PROGRAM PRG_SL2L0_POWER
VAR
	fbMotion1: FB_SimMotor;
	fbMotion2: FB_SimMotor;
	fbMotion3: FB_SimMotor;
	fbMotion4: FB_SimMotor;
END_VAR

// Placeholder, standard simulated motion for all axes
fbMotion1(stMotionStage := Main.M45);
fbMotion2(stMotionStage := Main.M46);
fbMotion3(stMotionStage := Main.M47);
fbMotion4(stMotionStage := Main.M48);

END_PROGRAM

(* stored: Version 1.1.0.1, ProductVersion 3.1.4022.12
   POU PRG_SL2L0_POWER: Id {b81ede99-2259-4f9f-b687-2b775d0f5c19}, SpecialFunc None *)
